Staubli VAL3: onInsert.pgx

public program onInsert(string& x_sItem[])
  local string l_sItem
  local string l_sEvent
  local num l_nSize
  local num l_nKey
begin
  //
  // compose the string
  // call getType(l_sItem)
  // x_sItem=l_sItem+" ???"
  //
  // insert all the saveAxis value from the list
  cls()
  call language:message(l_sEvent,65)
  call use:clear(0,13)
  call use:typeCenter(13,l_sEvent,40,true)
  x_sItem=""
  call use:setSizeList(19,0,19,10)
  call use:listcreate("AXIS7")
  l_nSize=size(nSaveaxis)
  for i=0 to l_nSize-1
    l_sEvent=sSaveaxis[i]
    call use:listadd(l_sEvent)
  endFor
  call use:listupdate(0)
  do
    l_nKey=getKey()
    call use:listevent(l_nKey,i,l_sEvent)
    delay(0)
  until l_nKey==255 or l_nKey==270
  if l_nKey==270
    x_sItem="AXIS7>"+l_sEvent
  endIf
  call use:nullKey(l_nKey)
  delay(0)
end
